ABB RobotStudio station: Escritura.rsstnx

Station Escritura (saved by RobotStudio 22.2.9947.0)
Controller Controller1
  mechanical unit ROB_1: IRB140_6_81_C_03, 6 joints, base frame (0, 0, 0) mm
Layout (positions relative to the parent item):
  - IRB140_6_81_C_03 [mechanism, from Robots\IRB140_6_81_C_G_03.rslib] at (0, 0, 0) mm; joint values [0.0585, 0.6088, 0.529, 1.2458, 0.8822, 2.1442] (rad or m)
  - Escritura_2 [part] at (300, 500, 0) mm, rotated rx 90 ry 0 rz -90 deg, size 412 x 219.1 x 283 mm
  - marcador [mechanism, from LibreriaRS\marcador.rslib] at (434.57, 73.09, 258.17) mm, rotated rx -132.86 ry 0 rz 0 deg
Attachment: marcador is attached to IRB140_6_81_C_03 / Link6
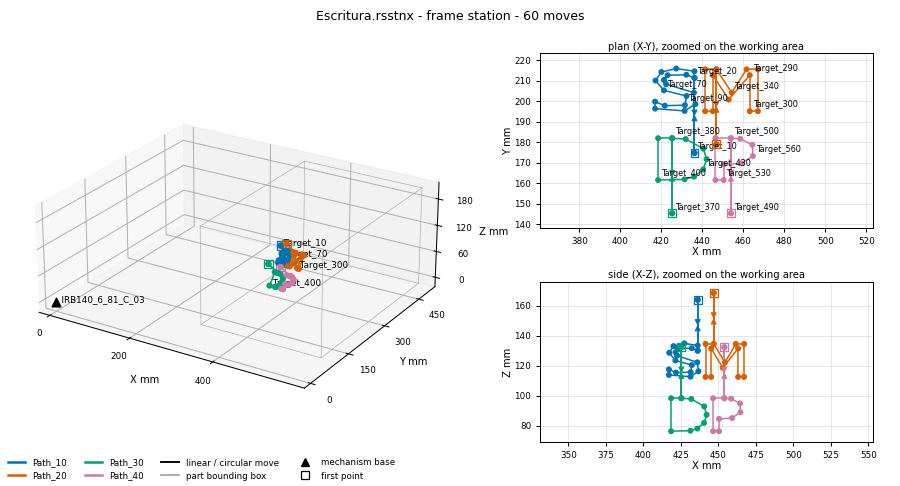
[picture p0: tool path of Escritura.rsstnx in frame station, 60 of 60 moves have a stored position in this frame; points joined in program order, loops and branches not executed]
Targets, tools, work objects and paths stored in the station, written as RAPID:
! task T_ROB1
MODULE CalibData
  PERS tooldata marcador:=[TRUE,[[1.646,0,138.55],[1,0,0,0]],[0.1,[0,0,44],[1,0,0,0],0,0,0]];
  TASK PERS wobjdata tablero283:=[FALSE,TRUE,"",[[0,0,0],[1,0,0,0]],[[0,0,0],[1,0,0,0]]];
ENDMODULE

! task T_ROB1
MODULE Module1
  CONST robtarget Target_10:=[[436.217949836,174.647221187,163.925939958],[0.399843528,-0.916583413,0,0],[0,0,0,0],[9E+09,9E+09,9E+09,9E+09,9E+09,9E+09]];
  CONST robtarget Target_20:=[[436.217949836,211.296215765,129.913424667],[0.399843528,-0.916583413,0,0],[0,0,0,0],[9E+09,9E+09,9E+09,9E+09,9E+09,9E+09]];
  CONST robtarget Target_30:=[[436.217949836,214.537602959,133.406067911],[0.399843528,-0.916583413,0,0],[0,0,0,0],[9E+09,9E+09,9E+09,9E+09,9E+09,9E+09]];
  CONST robtarget Target_40:=[[427.295745622,215.860618141,134.831636581],[0.399843528,-0.916583413,0,0],[0,0,0,0],[9E+09,9E+09,9E+09,9E+09,9E+09,9E+09]];
  CONST robtarget Target_50:=[[420.051013045,214.182042629,133.02294633],[0.399843528,-0.916583413,0,0],[0,0,0,0],[9E+09,9E+09,9E+09,9E+09,9E+09,9E+09]];
  CONST robtarget Target_60:=[[417.206604617,210.022813652,128.541314822],[0.399843528,-0.916583413,0,0],[0,0,0,0],[9E+09,9E+09,9E+09,9E+09,9E+09,9E+09]];
  CONST robtarget Target_70:=[[421.32735016,205.235152464,123.382538194],[0.399843528,-0.916583413,0,0],[0,0,0,0],[9E+09,9E+09,9E+09,9E+09,9E+09,9E+09]];
  CONST robtarget Target_80:=[[432.340316124,202.465089428,120.39775379],[0.399843528,-0.916583413,0,0],[0,0,0,0],[9E+09,9E+09,9E+09,9E+09,9E+09,9E+09]];
  CONST robtarget Target_90:=[[431.538047081,198.008182035,115.59536933],[0.399843528,-0.916583413,0,0],[0,0,0,0],[9E+09,9E+09,9E+09,9E+09,9E+09,9E+09]];
  CONST robtarget Target_100:=[[421.740640274,197.768385534,115.336985009],[0.399843528,-0.916583413,0,0],[0,0,0,0],[9E+09,9E+09,9E+09,9E+09,9E+09,9E+09]];
  CONST robtarget Target_110:=[[416.987803969,199.719832926,117.439698798],[0.399843528,-0.916583413,0,0],[0,0,0,0],[9E+09,9E+09,9E+09,9E+09,9E+09,9E+09]];
  CONST robtarget Target_120:=[[416.987803969,196.313068834,113.768859471],[0.399843528,-0.916583413,0,0],[0,0,0,0],[9E+09,9E+09,9E+09,9E+09,9E+09,9E+09]];
  CONST robtarget Target_130:=[[431.404335573,195.20504362,112.574945709],[0.399843528,-0.916583413,0,0],[0,0,0,0],[9E+09,9E+09,9E+09,9E+09,9E+09,9E+09]];
  CONST robtarget Target_140:=[[436.667706724,198.545656953,116.174506603],[0.399843528,-0.916583413,0,0],[0,0,0,0],[9E+09,9E+09,9E+09,9E+09,9E+09,9E+09]];
  CONST robtarget Target_150:=[[435.950526821,204.11058956,122.170804824],[0.399843528,-0.916583413,0,0],[0,0,0,0],[9E+09,9E+09,9E+09,9E+09,9E+09,9E+09]];
  CONST robtarget Target_160:=[[422.372731035,208.245012002,126.62570692],[0.399843528,-0.916583413,0,0],[0,0,0,0],[9E+09,9E+09,9E+09,9E+09,9E+09,9E+09]];
  CONST robtarget Target_170:=[[421.363816935,210.303954378,128.844248164],[0.399843528,-0.916583413,0,0],[0,0,0,0],[9E+09,9E+09,9E+09,9E+09,9E+09,9E+09]];
  CONST robtarget Target_180:=[[423.077755347,212.627499791,131.347903142],[0.399843528,-0.916583413,0,0],[0,0,0,0],[9E+09,9E+09,9E+09,9E+09,9E+09,9E+09]];
  CONST robtarget Target_190:=[[432.255226983,212.850758603,131.588467855],[0.399843528,-0.916583413,0,0],[0,0,0,0],[9E+09,9E+09,9E+09,9E+09,9E+09,9E+09]];
  CONST robtarget Target_200:=[[436.217949836,211.296215765,129.913424667],[0.399843528,-0.916583413,0,0],[0,0,0,0],[9E+09,9E+09,9E+09,9E+09,9E+09,9E+09]];
  CONST robtarget Target_210:=[[436.217949836,174.647221187,163.925939958],[0.399843528,-0.916583413,0,0],[0,0,0,0],[9E+09,9E+09,9E+09,9E+09,9E+09,9E+09]];
  CONST robtarget Target_220:=[[446.890559236,178.847794388,168.452120488],[0.399843528,-0.916583413,0,0],[0,0,0,0],[9E+09,9E+09,9E+09,9E+09,9E+09,9E+09]];
  CONST robtarget Target_230:=[[446.890559236,215.496788966,134.439605197],[0.399843528,-0.916583413,0,0],[0,0,0,0],[9E+09,9E+09,9E+09,9E+09,9E+09,9E+09]];
  CONST robtarget Target_240:=[[441.444854212,215.496788966,134.439605197],[0.399843528,-0.916583413,0,0],[0,0,0,0],[9E+09,9E+09,9E+09,9E+09,9E+09,9E+09]];
  CONST robtarget Target_250:=[[441.444854212,195.089279791,112.45020845],[0.399843528,-0.916583413,0,0],[0,0,0,0],[9E+09,9E+09,9E+09,9E+09,9E+09,9E+09]];
  CONST robtarget Target_260:=[[445.164465233,195.089279791,112.45020845],[0.399843528,-0.916583413,0,0],[0,0,0,0],[9E+09,9E+09,9E+09,9E+09,9E+09,9E+09]];
  CONST robtarget Target_270:=[[445.164465233,212.668844015,131.392452163],[0.399843528,-0.916583413,0,0],[0,0,0,0],[9E+09,9E+09,9E+09,9E+09,9E+09,9E+09]];
  CONST robtarget Target_280:=[[452.919732656,200.712094313,118.508875301],[0.399843528,-0.916583413,0,0],[0,0,0,0],[9E+09,9E+09,9E+09,9E+09,9E+09,9E+09]];
  CONST robtarget Target_290:=[[463.179051943,212.668844015,131.392452163],[0.399843529,-0.916583413,0,0],[0,0,0,0],[9E+09,9E+09,9E+09,9E+09,9E+09,9E+09]];
  CONST robtarget Target_300:=[[463.179051943,195.089279791,112.45020845],[0.399843528,-0.916583413,0,0],[0,0,0,0],[9E+09,9E+09,9E+09,9E+09,9E+09,9E+09]];
  CONST robtarget Target_310:=[[467.166085979,195.089279791,112.45020845],[0.399843528,-0.916583413,0,0],[0,0,0,0],[9E+09,9E+09,9E+09,9E+09,9E+09,9E+09]];
  CONST robtarget Target_320:=[[467.166085979,215.496788966,134.439605197],[0.399843528,-0.916583413,0,0],[0,0,0,0],[9E+09,9E+09,9E+09,9E+09,9E+09,9E+09]];
  CONST robtarget Target_330:=[[461.623136222,215.496788966,134.439605197],[0.399843528,-0.916583413,0,0],[0,0,0,0],[9E+09,9E+09,9E+09,9E+09,9E+09,9E+09]];
  CONST robtarget Target_340:=[[454.378403645,204.135396095,122.197534237],[0.399843529,-0.916583413,0,0],[0,0,0,0],[9E+09,9E+09,9E+09,9E+09,9E+09,9E+09]];
  CONST robtarget Target_350:=[[446.890559236,215.496788966,134.439605197],[0.399843528,-0.916583413,0,0],[0,0,0,0],[9E+09,9E+09,9E+09,9E+09,9E+09,9E+09]];
  CONST robtarget Target_360:=[[446.890559236,178.847794388,168.452120488],[0.399843528,-0.916583413,0,0],[0,0,0,0],[9E+09,9E+09,9E+09,9E+09,9E+09,9E+09]];
  CONST robtarget Target_370:=[[425.302228604,145.247366726,132.247156502],[0.399843528,-0.916583413,0,0],[0,0,0,0],[9E+09,9E+09,9E+09,9E+09,9E+09,9E+09]];
  CONST robtarget Target_380:=[[425.302228604,181.896361304,98.234641211],[0.399843528,-0.916583413,0,0],[0,0,0,0],[9E+09,9E+09,9E+09,9E+09,9E+09,9E+09]];
  CONST robtarget Target_390:=[[418.470786141,181.896361304,98.234641211],[0.399843528,-0.916583413,0,0],[0,0,0,0],[9E+09,9E+09,9E+09,9E+09,9E+09,9E+09]];
  CONST robtarget Target_400:=[[418.470786141,161.488852129,76.245244464],[0.399843528,-0.916583413,0,0],[0,0,0,0],[9E+09,9E+09,9E+09,9E+09,9E+09,9E+09]];
  CONST robtarget Target_410:=[[431.367868799,161.819605925,76.601636632],[0.399843528,-0.916583413,0,0],[0,0,0,0],[9E+09,9E+09,9E+09,9E+09,9E+09,9E+09]];
  CONST robtarget Target_420:=[[435.999149188,163.126083416,78.009385694],[0.399843528,-0.916583413,0,0],[0,0,0,0],[9E+09,9E+09,9E+09,9E+09,9E+09,9E+09]];
  CONST robtarget Target_430:=[[440.460251295,166.632073647,81.787142672],[0.399843529,-0.916583413,0,0],[0,0,0,0],[9E+09,9E+09,9E+09,9E+09,9E+09,9E+09]];
  CONST robtarget Target_440:=[[442.12556734,171.676069027,87.222123229],[0.399843528,-0.916583413,0,0],[0,0,0,0],[9E+09,9E+09,9E+09,9E+09,9E+09,9E+09]];
  CONST robtarget Target_450:=[[440.533184844,176.8110217,92.755111633],[0.399843528,-0.916583413,0,0],[0,0,0,0],[9E+09,9E+09,9E+09,9E+09,9E+09,9E+09]];
  CONST robtarget Target_460:=[[431.939181603,181.46638137,97.771331393],[0.399843528,-0.916583413,0,0],[0,0,0,0],[9E+09,9E+09,9E+09,9E+09,9E+09,9E+09]];
  CONST robtarget Target_470:=[[425.302228604,181.896361304,98.234641211],[0.399843528,-0.916583413,0,0],[0,0,0,0],[9E+09,9E+09,9E+09,9E+09,9E+09,9E+09]];
  CONST robtarget Target_480:=[[425.302228604,145.247366726,132.247156502],[0.399843528,-0.916583413,0,0],[0,0,0,0],[9E+09,9E+09,9E+09,9E+09,9E+09,9E+09]];
  CONST robtarget Target_490:=[[453.989424714,145.247366726,132.247156502],[0.399843528,-0.916583413,0,0],[0,0,0,0],[9E+09,9E+09,9E+09,9E+09,9E+09,9E+09]];
  CONST robtarget Target_500:=[[453.989424714,181.896361304,98.234641211],[0.399843528,-0.916583413,0,0],[0,0,0,0],[9E+09,9E+09,9E+09,9E+09,9E+09,9E+09]];
  CONST robtarget Target_510:=[[446.45295794,181.896361304,98.234641211],[0.399843528,-0.916583413,0,0],[0,0,0,0],[9E+09,9E+09,9E+09,9E+09,9E+09,9E+09]];
  CONST robtarget Target_520:=[[446.45295794,161.488852129,76.245244464],[0.399843528,-0.916583413,0,0],[0,0,0,0],[9E+09,9E+09,9E+09,9E+09,9E+09,9E+09]];
  CONST robtarget Target_530:=[[450.439991975,161.488852129,76.245244464],[0.399843528,-0.916583413,0,0],[0,0,0,0],[9E+09,9E+09,9E+09,9E+09,9E+09,9E+09]];
  CONST robtarget Target_540:=[[450.439991975,169.096189423,84.442264321],[0.399843528,-0.916583413,0,0],[0,0,0,0],[9E+09,9E+09,9E+09,9E+09,9E+09,9E+09]];
  CONST robtarget Target_550:=[[459.131239949,169.63366434,85.021401594],[0.399843528,-0.916583413,0,0],[0,0,0,0],[9E+09,9E+09,9E+09,9E+09,9E+09,9E+09]];
  CONST robtarget Target_560:=[[464.722812073,173.230611865,88.897166417],[0.399843528,-0.916583413,0,0],[0,0,0,0],[9E+09,9E+09,9E+09,9E+09,9E+09,9E+09]];
  CONST robtarget Target_570:=[[464.46754465,178.646705264,94.733088163],[0.399843529,-0.916583413,0,0],[0,0,0,0],[9E+09,9E+09,9E+09,9E+09,9E+09,9E+09]];
  CONST robtarget Target_580:=[[458.535615962,181.598682888,97.91388826],[0.399843529,-0.916583413,0,0],[0,0,0,0],[9E+09,9E+09,9E+09,9E+09,9E+09,9E+09]];
  CONST robtarget Target_590:=[[453.989424714,181.896361304,98.234641211],[0.399843528,-0.916583413,0,0],[0,0,0,0],[9E+09,9E+09,9E+09,9E+09,9E+09,9E+09]];
  CONST robtarget Target_600:=[[453.989424714,145.247366726,132.247156502],[0.399843528,-0.916583413,0,0],[0,0,0,0],[9E+09,9E+09,9E+09,9E+09,9E+09,9E+09]];
  PROC Path_10()
    MoveL Target_10,v50,z50,marcador\WObj:=tablero283;
    MoveL Target_20,v50,z50,marcador\WObj:=tablero283;
    MoveL Target_30,v50,z50,marcador\WObj:=tablero283;
    MoveL Target_40,v50,z50,marcador\WObj:=tablero283;
    MoveL Target_50,v50,z50,marcador\WObj:=tablero283;
    MoveL Target_60,v50,z50,marcador\WObj:=tablero283;
    MoveL Target_70,v50,z50,marcador\WObj:=tablero283;
    MoveL Target_80,v50,z50,marcador\WObj:=tablero283;
    MoveL Target_90,v50,z50,marcador\WObj:=tablero283;
    MoveL Target_100,v50,z50,marcador\WObj:=tablero283;
    MoveL Target_110,v50,z50,marcador\WObj:=tablero283;
    MoveL Target_120,v50,z50,marcador\WObj:=tablero283;
    MoveL Target_130,v50,z50,marcador\WObj:=tablero283;
    MoveL Target_140,v50,z50,marcador\WObj:=tablero283;
    MoveL Target_150,v50,z50,marcador\WObj:=tablero283;
    MoveL Target_160,v50,z50,marcador\WObj:=tablero283;
    MoveL Target_170,v50,z50,marcador\WObj:=tablero283;
    MoveL Target_180,v50,z50,marcador\WObj:=tablero283;
    MoveL Target_190,v50,z50,marcador\WObj:=tablero283;
    MoveL Target_200,v50,z50,marcador\WObj:=tablero283;
    MoveL Target_210,v50,z50,marcador\WObj:=tablero283;
  ENDPROC
  PROC Path_20()
    MoveL Target_220,v1000,z100,marcador\WObj:=tablero283;
    MoveL Target_230,v1000,z100,marcador\WObj:=tablero283;
    MoveL Target_240,v1000,z100,marcador\WObj:=tablero283;
    MoveL Target_250,v1000,z100,marcador\WObj:=tablero283;
    MoveL Target_260,v1000,z100,marcador\WObj:=tablero283;
    MoveL Target_270,v1000,z100,marcador\WObj:=tablero283;
    MoveL Target_280,v1000,z100,marcador\WObj:=tablero283;
    MoveL Target_290,v1000,z100,marcador\WObj:=tablero283;
    MoveL Target_300,v1000,z100,marcador\WObj:=tablero283;
    MoveL Target_310,v1000,z100,marcador\WObj:=tablero283;
    MoveL Target_320,v1000,z100,marcador\WObj:=tablero283;
    MoveL Target_330,v1000,z100,marcador\WObj:=tablero283;
    MoveL Target_340,v1000,z100,marcador\WObj:=tablero283;
    MoveL Target_350,v1000,z100,marcador\WObj:=tablero283;
    MoveL Target_360,v1000,z100,marcador\WObj:=tablero283;
  ENDPROC
  PROC Path_30()
    MoveL Target_370,v1000,z100,marcador\WObj:=tablero283;
    MoveL Target_380,v1000,z100,marcador\WObj:=tablero283;
    MoveL Target_390,v1000,z100,marcador\WObj:=tablero283;
    MoveL Target_400,v1000,z100,marcador\WObj:=tablero283;
    MoveL Target_410,v1000,z100,marcador\WObj:=tablero283;
    MoveL Target_420,v1000,z100,marcador\WObj:=tablero283;
    MoveL Target_430,v1000,z100,marcador\WObj:=tablero283;
    MoveL Target_440,v1000,z100,marcador\WObj:=tablero283;
    MoveL Target_450,v1000,z100,marcador\WObj:=tablero283;
    MoveL Target_460,v1000,z100,marcador\WObj:=tablero283;
    MoveL Target_470,v1000,z100,marcador\WObj:=tablero283;
    MoveL Target_480,v1000,z100,marcador\WObj:=tablero283;
  ENDPROC
  PROC Path_40()
    MoveL Target_490,v1000,z100,marcador\WObj:=tablero283;
    MoveL Target_500,v1000,z100,marcador\WObj:=tablero283;
    MoveL Target_510,v1000,z100,marcador\WObj:=tablero283;
    MoveL Target_520,v1000,z100,marcador\WObj:=tablero283;
    MoveL Target_530,v1000,z100,marcador\WObj:=tablero283;
    MoveL Target_540,v1000,z100,marcador\WObj:=tablero283;
    MoveL Target_550,v1000,z100,marcador\WObj:=tablero283;
    MoveL Target_560,v1000,z100,marcador\WObj:=tablero283;
    MoveL Target_570,v1000,z100,marcador\WObj:=tablero283;
    MoveL Target_580,v1000,z100,marcador\WObj:=tablero283;
    MoveL Target_590,v1000,z100,marcador\WObj:=tablero283;
    MoveL Target_600,v1000,z100,marcador\WObj:=tablero283;
  ENDPROC
ENDMODULE

